VISUALIZATION CtrlBox  // 2x2
END_VISUALIZATION

(* stored: Version 1.1.0.1, ProductVersion 3.1.4024.12
   Visu CtrlBox: Id {7bd49a86-7a8c-4981-a55e-e70a044c7b04} *)
